{attribute addProperty BoxType "EL9540-0010-0016"}
{attribute addProperty Id "UndervoltageAT %I*BOOL811OvervoltageAT %I*BOOL812"}
{attribute addProperty CRC "2971883996"}
{attribute addProperty SizeInBites "16"}
{attribute addProperty SizeInBytes "2"}
TYPE Status_Up_B12359DC :
STRUCT
	{attribute addProperty Name "Undervoltage"}
	Undervoltage AT %I* : BOOL;
	{attribute addProperty Name "Overvoltage"}
	Overvoltage AT %I* : BOOL;
END_STRUCT
END_TYPE

(* stored: Version 1.2.0.0, ProductVersion 3.1.4024.9
   DUT Status_Up_B12359DC: Id {57210ed4-04d8-4a1e-bc84-0ecf692e2c3a} *)
